// TIA Portal V21 export
// export: Created 2026-08-11T14:59:46Z, ExportSetting WithDefaults
VAR_GLOBAL   // PLC tag table "Outputs"
   Infeed_Run AT %Q0.0 : Bool;   // Infeed conveyor - contactor coil
   Clamp_Open AT %Q0.1 : Bool;   // Part clamp - open coil
   Clamp_Close AT %Q0.2 : Bool;   // Part clamp - close coil
   Lift_Open AT %Q0.3 : Bool;   // Transfer lift - solenoid coil
   Outfeed_Run AT %Q0.4 : Bool;   // Outfeed conveyor drive - drive run/enable
END_VAR
